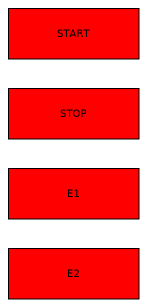
[picture p24: Zustaende (HMI screen)]
rounded rectangle at (50,0)-(181,51): text "START"; alarm colour if Ampelsteuerung.Start; taps Ampelsteuerung.Start
rounded rectangle at (50,80)-(181,131): text "STOP"; alarm colour if Ampelsteuerung.Stop; toggles Ampelsteuerung.Stop
rounded rectangle at (50,240)-(181,291): text "E2"; alarm colour if .E2
rounded rectangle at (50,160)-(181,211): text "E1"; alarm colour if .E1
*)
